// TIA Portal V17 export
// export: Created 2024-08-26T21:10:54.6916348Z, ExportSetting WithDefaults, DisplayName Totally Integrated Automation Portal, DisplayVersion V17 Update 7, DisplayName TIA Portal Openness, DisplayVersion V17 Update 7, DisplayName TIA Portal Version Control Interface, DisplayVersion V17, DisplayName SINAMICS Startdrive Advanced, DisplayVersion V17 SP2, DisplayName SINAMICS Startdrive G110M, G120, G120C, G120D, G120P, G115D, DisplayVersion V17 SP2, DisplayName SINAMICS Startdrive G130, G150, S120, S150, SINAMICS MV, S210, DisplayVersion V17 SP2, DisplayName STEP 7 Professional, DisplayVersion V17 Update 7, DisplayName STEP 7 Safety, DisplayVersion V17 Update 6, DisplayName WinCC Advanced / Unified PC, DisplayVersion V17 Update 7
TYPE "CONFIG_MSG_IJC"
// stored: IsFailsafeCompliant false
   STRUCT
      "TYPE" : String[3];
      KANBAN : String[30];
      COMPONENT : String[62];
      START : Bool;
      PROCESS_STATUS : SInt;
   END_STRUCT;
END_TYPE
